TYPE User:
	STRUCT
		UserID: INT;
		UserNumber: STRING;
		UserName: STRING;
		UserLevel: INT;
		UserExist: BOOL;
	END_STRUCT
END_TYPE

(* stored: Version 1.1.0.1, ProductVersion 3.1.4024.11
   DUT User: Id {38b2271d-160d-4879-a990-df1d4ac1584b} *)
